FUNCTION_BLOCK DeleteMe
VAR_INPUT
END_VAR
VAR_OUTPUT
END_VAR
VAR

END_VAR


(*  *********************************************************** *)
(*  Laborplatte Linearachse                                     *)
(*  *********************************************************** *)

DA.P1 := DI.S1;
DA.P2 := DI.S2;
DA.P3 := DI.S3;

DA.Q1 := DI.S4;
DA.Q2 := DI.S5;

END_FUNCTION_BLOCK

(* stored: Version 1.1.0.1, ProductVersion 3.1.4024.5
   POU DeleteMe: Id {f156885e-d892-4706-970d-8d2a74171c01}, SpecialFunc None *)
